FUNCTION TryConvert_ULINT_TO_DINT : BOOL
VAR_INPUT
	in : ULINT;
	out : REFERENCE TO DINT;
END_VAR

IF in > DatatypeLimits.MAX_VALUE_OF_ULINT_WHICH_CAN_BE_HELD_IN_A_DINT THEN
	RETURN;
END_IF

out := ULINT_TO_DINT(in);
TryConvert_ULINT_TO_DINT := TRUE;

END_FUNCTION

(* stored: Version 1.1.0.1, ProductVersion 3.1.4024.12
   POU TryConvert_ULINT_TO_DINT: Id {70fc584e-d76d-4cc3-93ff-0197d7b93726}, SpecialFunc None *)
